--- Backups/pr3/RAPID/TASK1/PROGMOD/Module1.mod ---
MODULE Module1
	CONST robtarget Target_10:=[[1359.914350434,189.052041228,1867.751078124],[0.28377426,-0.836118095,0.437820703,-0.169386341],[0,0,-3,0],[9E+09,9E+09,9E+09,9E+09,9E+09,9E+09]];
	CONST robtarget Target_20:=[[1359.914369628,120.392226788,1867.751087064],[0.283774546,-0.836118001,0.43782057,-0.169386668],[0,0,-3,0],[9E+09,9E+09,9E+09,9E+09,9E+09,9E+09]];
	CONST robtarget Target_30:=[[1359.914226872,120.392161677,1060.024906535],[0.283774755,-0.836117846,0.437820445,-0.169387409],[0,1,-3,0],[9E+09,9E+09,9E+09,9E+09,9E+09,9E+09]];
	CONST robtarget Target_40:=[[1288.339226949,142.88058846,1159.109938579],[0.283774905,-0.836117579,0.437820302,-0.169388845],[0,1,-3,0],[9E+09,9E+09,9E+09,9E+09,9E+09,9E+09]];
	CONST robtarget Target_50:=[[1288.339333488,142.880646916,1864.033074108],[0.283776583,-0.836117259,0.437818944,-0.169391124],[0,0,-3,0],[9E+09,9E+09,9E+09,9E+09,9E+09,9E+09]];
	CONST robtarget Target_60:=[[1396.622330981,211.05352138,1797.840056923],[0.283777308,-0.836116859,0.437818886,-0.169392034],[0,0,-3,0],[9E+09,9E+09,9E+09,9E+09,9E+09,9E+09]];
	CONST robtarget Target_70:=[[1225.907089757,47.887281808,1220.291013598],[0.283778703,-0.836117031,0.437817025,-0.169393657],[-1,1,-3,0],[9E+09,9E+09,9E+09,9E+09,9E+09,9E+09]];
	CONST robtarget Target_80:=[[1225.907079131,47.887238756,979.783968451],[0.283778643,-0.836116986,0.437817072,-0.169393858],[-1,1,-3,0],[9E+09,9E+09,9E+09,9E+09,9E+09,9E+09]];
	CONST robtarget Target_90:=[[1225.907179869,110.196868604,823.578395227],[0.283778412,-0.836116876,0.43781729,-0.169394225],[0,1,-4,0],[9E+09,9E+09,9E+09,9E+09,9E+09,9E+09]];
	CONST robtarget Target_100:=[[1035.260759077,110.196845363,823.578341268],[0.283778036,-0.836117118,0.437816894,-0.169394683],[0,1,-4,0],[9E+09,9E+09,9E+09,9E+09,9E+09,9E+09]];
	CONST robtarget Target_110:=[[1035.261060311,110.196778558,823.57799127],[0.341042108,-0.743784627,0.47971346,-0.316780217],[0,2,-4,0],[9E+09,9E+09,9E+09,9E+09,9E+09,9E+09]];
	CONST robtarget Target_120:=[[1035.2615814,110.19683868,823.577736078],[0.306762006,-0.695295218,0.550476721,-0.345596603],[0,3,-5,0],[9E+09,9E+09,9E+09,9E+09,9E+09,9E+09]];
	CONST robtarget Target_130:=[[1227.749003758,-87.086102015,898.637389106],[0.401803093,-0.83564632,0.29691234,-0.228237957],[-1,1,-4,0],[9E+09,9E+09,9E+09,9E+09,9E+09,9E+09]];
	CONST robtarget Target_140:=[[1247.926834673,-113.238805252,518.057828259],[0.401801987,-0.835647129,0.296911763,-0.228237691],[-1,2,-4,0],[9E+09,9E+09,9E+09,9E+09,9E+09,9E+09]];
	CONST robtarget Target_150:=[[1264.237758862,-145.855770141,241.966431846],[0.401801453,-0.835648597,0.296909613,-0.228236053],[-1,2,-4,0],[9E+09,9E+09,9E+09,9E+09,9E+09,9E+09]];
	CONST robtarget Target_160:=[[1128.0688239,-143.135341759,292.908969476],[0.401800911,-0.835651508,0.296904199,-0.228233393],[-1,2,-4,0],[9E+09,9E+09,9E+09,9E+09,9E+09,9E+09]];
	CONST robtarget Target_170:=[[1128.069049024,-143.135368985,729.590033266],[0.401800633,-0.835651641,0.296904229,-0.228233356],[-1,1,-4,0],[9E+09,9E+09,9E+09,9E+09,9E+09,9E+09]];
	CONST robtarget Target_180:=[[1236.096802902,-96.606788938,264.050379664],[0.844944992,-0.381876574,0.080734356,-0.365677736],[-1,1,-4,1],[9E+09,9E+09,9E+09,9E+09,9E+09,9E+09]];
	CONST robtarget Target_190:=[[1263.432163062,-49.076157559,219.686861759],[0.84494253,-0.381881448,0.080736569,-0.365677845],[-1,1,-4,1],[9E+09,9E+09,9E+09,9E+09,9E+09,9E+09]];
	CONST robtarget Target_200:=[[1237.348016113,-55.067728806,185.37023784],[0.844936834,-0.381892704,0.080740996,-0.365678275],[-1,1,-4,1],[9E+09,9E+09,9E+09,9E+09,9E+09,9E+09]];
	CONST robtarget Target_210:=[[1065.206110583,-52.115045672,185.369462943],[0.844935801,-0.38189476,0.080741711,-0.365678357],[-1,1,-4,1],[9E+09,9E+09,9E+09,9E+09,9E+09,9E+09]];
	CONST robtarget Target_220:=[[1218.03502948,-52.114690425,166.267960314],[0.844934253,-0.381898356,0.080742219,-0.365678066],[-1,1,-4,1],[9E+09,9E+09,9E+09,9E+09,9E+09,9E+09]];
	CONST robtarget Target_230:=[[1218.035057782,0.360283476,166.267597723],[0.844933777,-0.381899344,0.08074267,-0.365678035],[-1,1,-4,1],[9E+09,9E+09,9E+09,9E+09,9E+09,9E+09]];
	CONST robtarget Target_240:=[[1049.013112504,0.360320531,166.267173862],[0.844933246,-0.381900492,0.080742991,-0.365677991],[-1,1,-4,1],[9E+09,9E+09,9E+09,9E+09,9E+09,9E+09]];
	CONST robtarget Target_250:=[[741.479498812,21.487944281,460.641074795],[0.167046833,0.579624718,0.293347911,0.741672127],[-1,2,-5,1],[9E+09,9E+09,9E+09,9E+09,9E+09,9E+09]];
	CONST robtarget Target_260:=[[741.47959356,52.990017017,468.573399202],[0.167047709,0.579627016,0.293349084,0.741669671],[0,2,-5,1],[9E+09,9E+09,9E+09,9E+09,9E+09,9E+09]];
	CONST robtarget Target_270:=[[741.479470826,52.989743441,402.945757804],[0.167048259,0.579628065,0.293349195,0.741668683],[0,2,-5,1],[9E+09,9E+09,9E+09,9E+09,9E+09,9E+09]];
	CONST robtarget Target_280:=[[741.479437654,-21.578976222,402.945438683],[0.167047992,0.579628558,0.293349684,0.741668165],[-1,2,-5,1],[9E+09,9E+09,9E+09,9E+09,9E+09,9E+09]];
	CONST robtarget Target_290:=[[741.479455644,-21.579005192,495.449003725],[0.167047914,0.579629056,0.29334997,0.74166768],[-1,2,-5,1],[9E+09,9E+09,9E+09,9E+09,9E+09,9E+09]];
	CONST robtarget Target_300:=[[954.088201372,127.514709299,272.759250433],[0.167048682,0.579633756,0.293351441,0.741663252],[0,2,-5,1],[9E+09,9E+09,9E+09,9E+09,9E+09,9E+09]];
	CONST robtarget Target_310:=[[954.088095411,127.514510621,-13.446080114],[0.167048969,0.579635488,0.293351958,0.741661629],[0,2,-5,1],[9E+09,9E+09,9E+09,9E+09,9E+09,9E+09]];
	CONST robtarget Target_320:=[[954.087987294,42.729988075,-13.446422439],[0.167048805,0.579636058,0.293352405,0.741661043],[-1,2,-5,1],[9E+09,9E+09,9E+09,9E+09,9E+09,9E+09]];
	CONST robtarget Target_330:=[[954.087890772,42.72997271,305.664990545],[0.167048406,0.579637688,0.293353566,0.741659401],[-1,2,-5,1],[9E+09,9E+09,9E+09,9E+09,9E+09,9E+09]];
	CONST robtarget Target_340:=[[1062.705954522,42.729934145,305.664692576],[0.167048487,0.579638189,0.293353947,0.74165884],[-1,2,-5,1],[9E+09,9E+09,9E+09,9E+09,9E+09,9E+09]];
	CONST robtarget Target_350:=[[1062.705913046,42.729918606,-20.939554836],[0.167048412,0.579638718,0.293354285,0.74165831],[-1,2,-5,1],[9E+09,9E+09,9E+09,9E+09,9E+09,9E+09]];
	CONST robtarget Target_360:=[[1062.705922672,-42.780840866,-20.939905277],[0.167048299,0.579639297,0.293354716,0.741657712],[-1,2,-5,1],[9E+09,9E+09,9E+09,9E+09,9E+09,9E+09]];
	CONST robtarget Target_370:=[[1062.705963822,-42.780859644,358.539699735],[0.167048216,0.579639878,0.293354953,0.741657182],[-1,2,-5,0],[9E+09,9E+09,9E+09,9E+09,9E+09,9E+09]];
	PERS num ColorIndex3:=1;
    CONST robtarget Target_180_2:=[[1236.09620943,-229.253997693,264.04805571],[0.892729073,-0.435461507,-0.046433543,-0.10607546],[-1,1,-4,1],[9E+09,9E+09,9E+09,9E+09,9E+09,9E+09]];
    CONST robtarget Target_380:=[[1062.706013298,254.661882488,394.279567264],[0.022239678,-0.602825102,-0.047180566,-0.79616662],[0,2,-5,1],[9E+09,9E+09,9E+09,9E+09,9E+09,9E+09]];
    CONST robtarget Target_390:=[[729.42291728,228.831924059,394.278056221],[0.022236675,-0.602828487,-0.047179166,-0.796164224],[0,2,-5,1],[9E+09,9E+09,9E+09,9E+09,9E+09,9E+09]];
    CONST robtarget Target_400:=[[992.762340696,228.831189854,180.25404409],[0.022234595,-0.602832885,-0.047178666,-0.796160982],[0,2,-5,1],[9E+09,9E+09,9E+09,9E+09,9E+09,9E+09]];
    CONST robtarget Target_410:=[[992.76307458,129.831933881,781.600340796],[0.005972285,-0.914865356,0.069810272,-0.397633295],[0,3,-6,0],[9E+09,9E+09,9E+09,9E+09,9E+09,9E+09]];
    CONST robtarget Target_420:=[[1274.891703819,171.05584658,1014.941903815],[0.005970392,-0.91486556,0.069814373,-0.397632135],[0,4,-6,0],[9E+09,9E+09,9E+09,9E+09,9E+09,9E+09]];
    CONST robtarget Target_430:=[[1047.127100193,89.200489047,835.063488807],[0.001681943,0.952786124,-0.070049154,0.295446931],[0,4,-7,0],[9E+09,9E+09,9E+09,9E+09,9E+09,9E+09]];
    PROC Path_10()
        ColorIndex3:=1;
        Set do3;
        WaitTime 1;
	    MoveL Target_10,v500,fine,tool0\WObj:=wobj0;
	    MoveL Target_20,v500,fine,tool0\WObj:=wobj0;
	    MoveL Target_30,v500,fine,tool0\WObj:=wobj0;
	    MoveL Target_40,v500,fine,tool0\WObj:=wobj0;
	    MoveL Target_50,v500,fine,tool0\WObj:=wobj0;
	    MoveL Target_60,v500,fine,tool0\WObj:=wobj0;
	    MoveL Target_70,v500,fine,tool0\WObj:=wobj0;
	    MoveL Target_80,v500,fine,tool0\WObj:=wobj0;
	    MoveL Target_90,v500,fine,tool0\WObj:=wobj0;
	    MoveL Target_100,v500,fine,tool0\WObj:=wobj0;
	    MoveL Target_110,v500,fine,tool0\WObj:=wobj0;
	    MoveL Target_120,v500,fine,tool0\WObj:=wobj0;
	    MoveL Target_130,v500,fine,tool0\WObj:=wobj0;
	    MoveL Target_140,v500,fine,tool0\WObj:=wobj0;
	    MoveL Target_150,v500,fine,tool0\WObj:=wobj0;
	    MoveL Target_160,v500,fine,tool0\WObj:=wobj0;
	    MoveL Target_170,v500,fine,tool0\WObj:=wobj0;
	    MoveL Target_180,v500,fine,tool0\WObj:=wobj0;
	    MoveL Target_180_2,v500,fine,tool0\WObj:=wobj0;
	    MoveL Target_180,v500,fine,tool0\WObj:=wobj0;
	    MoveL Target_190,v500,fine,tool0\WObj:=wobj0;
	    MoveL Target_200,v500,fine,tool0\WObj:=wobj0;
	    MoveL Target_210,v500,fine,tool0\WObj:=wobj0;
	    MoveL Target_220,v500,fine,tool0\WObj:=wobj0;
	    MoveL Target_230,v500,fine,tool0\WObj:=wobj0;
	    MoveL Target_240,v500,fine,tool0\WObj:=wobj0;
	    MoveL Target_250,v500,fine,tool0\WObj:=wobj0;
	    MoveL Target_260,v500,fine,tool0\WObj:=wobj0;
	    MoveL Target_270,v500,fine,tool0\WObj:=wobj0;
	    MoveL Target_280,v500,fine,tool0\WObj:=wobj0;
	    MoveL Target_290,v500,fine,tool0\WObj:=wobj0;
	    MoveL Target_310,v500,fine,tool0\WObj:=wobj0;
	    MoveL Target_320,v500,fine,tool0\WObj:=wobj0;
	    MoveL Target_330,v500,fine,tool0\WObj:=wobj0;
	    MoveL Target_350,v500,fine,tool0\WObj:=wobj0;
	    MoveL Target_360,v500,fine,tool0\WObj:=wobj0;
	    MoveL Target_370,v500,fine,tool0\WObj:=wobj0;
        MoveL Target_380,v500,fine,tool0\WObj:=wobj0;
        MoveL Target_390,v500,fine,tool0\WObj:=wobj0;
        MoveL Target_400,v1000,z100,tool0\WObj:=wobj0;
        MoveL Target_410,v1000,z100,tool0\WObj:=wobj0;
        MoveL Target_420,v1000,fine,tool0\WObj:=wobj0;
        MoveL Target_430,v1000,fine,tool0\WObj:=wobj0;
        WaitTime 1;
        Reset do3;
	ENDPROC
ENDMODULE

--- Backups/pr1/HOME/programs/calpos.mod ---
module calpos

   ! SCOPE: Universal calibration/sync position program.

   proc mainCalPos()
      var jointtarget jLocalCalPos;

      ! Dummy instruction for SetPP.
      WaitTime 1;

      ! Set default values for all axis.
      jLocalCalPos := [[9E+09,9E+09,9E+09,9E+09,9E+09,9E+09],[9E+09,9E+09,9E+09,9E+09,9E+09,0]];

      jLocalCalPos.robax.rax_1 := nArmCalPos("rob1_1");
      jLocalCalPos.robax.rax_2 := nArmCalPos("rob1_2");
      jLocalCalPos.robax.rax_3 := nArmCalPos("rob1_3");
      jLocalCalPos.robax.rax_4 := nArmCalPos("rob1_4");
      jLocalCalPos.robax.rax_5 := nArmCalPos("rob1_5");
      jLocalCalPos.robax.rax_6 := nArmCalPos("rob1_6");

      if nRobSerialPart() = 5500 or nRobSerialPart() = 5510 then
         ! IRB5500 and IRB5510 has special values on axis 5 and 6, just set to 0 as stated in the manual.
         jLocalCalPos.robax.rax_5 := 0;
         jLocalCalPos.robax.rax_6 := 0;
      endif

      if stSingleJoint("AX7_1") <> "" then
         ! 7-axis robot.
         jLocalCalPos.extax.eax_a := nArmCalPos(stSingleJoint("AX7_1") \NoConversion)*1000;
      elseif nArmCalPos("obp_3") <> 9E+09 then
         ! 3-axis TurnTable.
         !IndReset OBP,2\RefNum:=0\Short;
         !IndReset OBP,3\RefNum:=0\Short;
         jLocalCalPos.extax.eax_a := nArmCalPos("obp_1");
         jLocalCalPos.extax.eax_b := nArmCalPos("obp_2");
         jLocalCalPos.extax.eax_c := nArmCalPos("obp_3");
      elseif nArmCalPos("obp_2") <> 9E+09 then
         ! 2-axis TurnTable.
         jLocalCalPos.extax.eax_a := nArmCalPos("obp_1");
         jLocalCalPos.extax.eax_b := nArmCalPos("obp_2");
      elseif nArmCalPos("obp_1") <> 9E+09 then
         ! 1-axis TurnTable.
         jLocalCalPos.extax.eax_a := nArmCalPos("obp_1");
      elseif nArmCalPos("track1") <> 9E+09 then
         ! IRB5350-02.
         jLocalCalPos.robax.rax_4 := 0;
         jLocalCalPos.robax.rax_5 := 0;
         jLocalCalPos.robax.rax_6 := 0;
         jLocalCalPos.extax.eax_a := nArmCalPos("track1" \NoConversion);
      elseif stRobotType() = "ROB1_5350_01_T00F82_A21C21D21" then
         ! IRB5350-01.
         jLocalCalPos.robax.rax_4 := 0;
         jLocalCalPos.robax.rax_5 := 0;
         jLocalCalPos.robax.rax_6 := 0;
      else
         ! Attempt to get values for 8-axis robot.
         jLocalCalPos.extax.eax_a := nArmCalPos("rob1_7" \NoConversion);
         jLocalCalPos.extax.eax_b := nArmCalPos("rob1_8" \NoConversion);
      endif

      if stSingleJoint("H1AngleAxis") <> "" then
         ! Global CBS.
         jLocalCalPos.extax.eax_b := 0;
         jLocalCalPos.extax.eax_c := 0;
         jLocalCalPos.extax.eax_d := 0;
         jLocalCalPos.extax.eax_e := 0;
      endif

      MoveAbsJ jLocalCalPos,v100,fine,tool0;
      Stop;
   endproc

   local func num nArmCalPos(string stArm \switch NoConversion)
      var num nCalPos;
      ReadCfgData "/MOC/ARM/" + stArm, "cal_position", nCalPos;
      if Present(NoConversion) then
         return nCalPos;
      else
         return Round(nCalPos * (180 / 3.1415926) \Dec := 3);
      endif
   error
      if errno = ERR_CFG_NOTFND then
         SkipWarn;
         return 9E+09;
      endif
   endfunc

   local func string stSingleJoint(string stSingle)
      var string stJoint;
      ReadCfgData "/MOC/SINGLE/" + stSingle, "use_joint", stJoint;
      return stJoint;
   error
      if errno = ERR_CFG_NOTFND then
         SkipWarn;
         return "";
      endif
   endfunc

   local func num nRobSerialPart()
      var string stPart;
      var num nPart;
      ReadCfgData "/MOC/ROBOT_SERIAL_NUMBER/PID", "robot_serial_number_high_part", stPart;
      if StrToVal(StrPart(stPart, 1, StrFind(stPart, 1, "_") - 1), nPart) then
         return nPart;
      else
         return 9E+09;
      endif
   error
      SkipWarn;
      return 9E+09;
   endfunc

   local func string stRobotType()
      var string stType;
      ReadCfgData "/MOC/ROBOT/ROB_1", "use_robot_type", stType;
      return stType;
   error
      if errno = ERR_CFG_NOTFND then
         SkipWarn;
         return "";
      endif
   endfunc

endmodule

--- Backups/pr1/HOME/programs/m1.mod ---
MODULE M1

  PROC mainM1()
    WaitTime 10;
  ENDPROC

ENDMODULE

--- Backups/pr1/HOME/programs/m10001.mod ---
module m10001

   ! SCOPE: Motion program for home position.

   proc mainm10001()
      if jHomePos.robax.rax_1 = 9E+09 then
         ErrWrite \W, "Home position not taught!", "";
      else
         MoveAbsJ jHomePos,v300,fine,tUserTool0;
      endif
   endproc

endmodule

--- Backups/pr1/HOME/programs/m2.mod ---
MODULE M2

  PROC mainM2()
    WaitTime 10;
  ENDPROC

ENDMODULE

--- Backups/pr1/HOME/programs/m3.mod ---
MODULE M3

  PROC mainM3()
    WaitTime 10;
  ENDPROC

ENDMODULE

--- Backups/pr1/SYSPAR/EIO.cfg ---
EIO:CFG_1.0:6:1::
#
SYSSIG_OUT:

      -Status "AutoOn" -Signal "AutoModeOn"

      -Status "RunchOk" -Signal "RunChainClosed"

      -Status "Error" -Signal "sdoRobotError"

      -Status "CycleOn" -Signal "sdoCycleOn"

      -Status "EmStop" -Signal "EmergencyStop"

      -Status "MotOnState" -Signal "MotorIsOn"

      -Status "WriteAccess" -Signal "MasterGranted"

      -Status "MotSupTrigg" -Signal "MotionSupTrigg"
#
SYSSIG_IN:

      -Signal "sdoAckAutoMode" -Action "AckAutoMode"

      -Signal "sdoResetError" -Action "ResetError"

      -Signal "sdoStartMain" -Action "StartMain"

      -Signal "sdoMotOnStart" -Action "MotOnStart"

      -Signal "sdoStop" -Action "Stop"

      -Signal "sdoQuickStop" -Action "QuickStop"

      -Signal "sdoMotorOn" -Action "MotorOn"

      -Signal "sdoMotorOff" -Action "MotorOff"

      -Signal "sdoWriteRequest" -Action "WriteAccess"
#
INDUSTRIAL_NETWORK:

      -Name "DeviceNet" -Label "DeviceNet Master/Slave Network" -Address "2"
#
EIO_CROSS:

      -Name "ReadyToReceiveCross" -Res "ReadyToReceive" -Act1 "doQueueFull"\
      -Act1_invert

      -Name "JobPendingCross" -Res "JobPending" -Act1 "doQueueEmpty"\
      -Act1_invert

      -Name "MtrlChRunningCross" -Res "MtrlChRunning" -Act1 "doMCSuspended"\
      -Act1_invert

      -Name "AppEnabledCross" -Res "AppEnabled" -Act1 "A1Enable"

      -Name "AppErrorCross" -Res "AppError" -Act1 "A1Error"

      -Name "HVEnabledCross" -Res "HVEnabled" -Act1 "A1HVEn" -Oper1 "AND"\
      -Act2 "READY_HV_ON"

      -Name "PotLifeWarningCross" -Res "PotLifeWarning" -Act1 "A1FluidPlWS"

      -Name "PotLifeTimeOutCross" -Res "PotLifeTimeOut" -Act1 "A1FluidPlTO"

      -Name "HomePosCross" -Res "HomePos" -Act1 "doHomePos"

      -Name "MtrlChangePosCross" -Res "MtrlChangePos" -Act1 "doMtrlChangePos"

      -Name "ReadyPosCross" -Res "ReadyPos" -Act1 "doReadyPos"

      -Name "UserPosCross" -Res "UserPos" -Act1 "doUserPos"

      -Name "doSwitchInAutoCross" -Res "doSwitchInAuto" -Act1 "AUTO1"\
      -Oper1 "AND" -Act2 "AUTO2"

      -Name "GoingToAutoCross" -Res "GoingToAuto" -Act1 "doSwitchInAuto"\
      -Oper1 "AND" -Act2 "AutoModeOn" -Act2_invert

      -Name "ReadyHighPriCross" -Res "ReadyHighPri" -Act1 "sdoCycleOn"\
      -Oper1 "AND" -Act2 "JobInProgress" -Act2_invert

      -Name "SystemRunningCross" -Res "SystemRunning" -Act1 "sdoCycleOn"\
      -Oper1 "AND" -Act2 "doQueuePause" -Act2_invert

      -Name "RobotErrorCross" -Res "RobotError" -Act1 "sdoRobotError"\
      -Oper1 "OR" -Act2 "doPntRapidError"

      -Name "BellRotatingCross" -Res "BellRotating" -Act1 "A1BellRotating"
#
DEVICENET_INTERNAL_DEVICE:

      -Name "DN_Internal_Device" -VendorName "ABB Robotics"\
      -ProductName "DeviceNet Internal Slave Device"
#
ICI_DEVICE:

      -Name "PIB" -Network "ICI" -Label "Process Interface Board"\
      -Address "192.168.126.200"
#
EIO_SIGNAL:

      -Name "AutoModeOn" -SignalType "DO"

      -Name "MasterGranted" -SignalType "DO"

      -Name "RunChainClosed" -SignalType "DO"

      -Name "RobotError" -SignalType "DO"

      -Name "JobInProgress" -SignalType "DO"

      -Name "JobPending" -SignalType "DO"

      -Name "ReadyHighPri" -SignalType "DO"

      -Name "SystemRunning" -SignalType "DO"

      -Name "MtrlChRunning" -SignalType "DO"

      -Name "MtrlChangeOn" -SignalType "DO"

      -Name "ObjConnected" -SignalType "DO"

      -Name "MtrlSupplyError" -SignalType "DO"

      -Name "AppEnabled" -SignalType "DO"

      -Name "AppError" -SignalType "DO"

      -Name "HVEnabled" -SignalType "DO"

      -Name "HVError" -SignalType "DO"

      -Name "PotLifeWarning" -SignalType "DO"

      -Name "PotLifeTimeOut" -SignalType "DO"

      -Name "HomePos" -SignalType "DO"

      -Name "MtrlChangePos" -SignalType "DO"

      -Name "ReadyPos" -SignalType "DO"

      -Name "UserPos" -SignalType "DO"

      -Name "ReposFinished" -SignalType "DO"

      -Name "EmergencyStop" -SignalType "DO"

      -Name "JobComplete" -SignalType "DO"

      -Name "GoingToAuto" -SignalType "DO"

      -Name "ReadyToReceive" -SignalType "DO"

      -Name "MotorIsOn" -SignalType "DO"

      -Name "ConveyorRunning" -SignalType "DO"

      -Name "ProgramLoaded" -SignalType "DO"

      -Name "CBSMotorIsOn" -SignalType "DO"

      -Name "BellRotating" -SignalType "DO"

      -Name "MotionSupTrigg" -SignalType "DO"

      -Name "doQueueFull" -SignalType "DO"

      -Name "doQueueEmpty" -SignalType "DO"

      -Name "doQueuePause" -SignalType "DO"

      -Name "doInModule" -SignalType "DO"

      -Name "doMCSuspended" -SignalType "DO"

      -Name "A1Enable" -SignalType "DO" -Access "All"

      -Name "A1Error" -SignalType "DO" -Access "All"

      -Name "A1HVEn" -SignalType "DO" -Access "All"

      -Name "A1FluidPlWS" -SignalType "DO" -Access "All"

      -Name "A1FluidPlTO" -SignalType "DO" -Access "All"

      -Name "doHomePos" -SignalType "DO" -Access "ReadOnly"

      -Name "doMtrlChangePos" -SignalType "DO" -Access "ReadOnly"

      -Name "doReadyPos" -SignalType "DO" -Access "ReadOnly"

      -Name "doUserPos" -SignalType "DO" -Access "ReadOnly"

      -Name "doSwitchInAuto" -SignalType "DO"

      -Name "doPntRapidError" -SignalType "DO"

      -Name "sdoRobotError" -SignalType "DO"

      -Name "sdoAckAutoMode" -SignalType "DO"

      -Name "sdoResetError" -SignalType "DO"

      -Name "sdoStartMain" -SignalType "DO"

      -Name "sdoMotOnStart" -SignalType "DO"

      -Name "sdoStop" -SignalType "DO"

      -Name "sdoQuickStop" -SignalType "DO"

      -Name "sdoMotorOn" -SignalType "DO"

      -Name "sdoMotorOff" -SignalType "DO"

      -Name "sdoCycleOn" -SignalType "DO"

      -Name "sdoWriteRequest" -SignalType "DO"

      -Name "A1Brush" -SignalType "GO" -Access "All"

      -Name "A1BrushTabNdx" -SignalType "GO" -Access "All"

      -Name "A1HVErrNo" -SignalType "GO" -Access "All"

      -Name "A1Material" -SignalType "GO" -Access "All"

      -Name "A1Fluid" -SignalType "AO" -Access "All"

      -Name "A1FluidAccu" -SignalType "AO" -Access "All"

      -Name "A1FluidEn" -SignalType "DO" -Access "All"

      -Name "A1NeedleEn" -SignalType "DO" -Access "All"

      -Name "A1BellRotating" -SignalType "DI" -Access "All"

      -Name "A1BrushTabLimEn" -SignalType "DO" -Access "All"

      -Name "do1" -SignalType "DO"

--- Backups/pr1/SYSPAR/PROC.cfg ---
PROC:CFG_1.0:6:0::
#
PW_SYSTEM:

      -name "PW_SYS" -pw_function "PW_FUNC"
#
PW_FUNCTION:

      -name "PW_FUNC" -do_repos_finished "ReposFinished"
#
PW_SERVICES_CONFIG:

      -Name "ProgramDirectory" -Value "HOME:/programs/"

      -Name "ProgramCache" -Value "False"

      -Name "LoadFailureModule" -Value ""

      -Name "ProgramStaticLoad" -Value "False"

      -Name "ProgramBackupSave" -Value "False"

      -Name "ProdLogDirectory" -Value "HOME:/logs"

      -Name "ProdLogFormat"\
      -Value "%D,Prog:%P,Mtrl:%M,Brush:%B,Usage:%C,CycleTime:%T"

      -Name "ProdLogSize" -Value "100000"

      -Name "JobQueueSize" -Value "10"

      -Name "JobQueueSave" -Value "False"

      -Name "JobQueueExpediteBegin" -Value "10001"

      -Name "JobQueueExpediteEnd" -Value "10016"

      -Name "ProgramIndexFile" -Value "HOME:/programs/segments.ndx"

      -Name "ExternalStart" -Value "False"

      -Name "JobQueueIgnoreMaterial" -Value "True"

      -Name "TipCleanModule" -Value "TipClean"

      -Name "TipCleanInterval" -Value "0"

      -Name "TipCleanModuleFile" -Value ""

      -Name "TipCleanIntervalFile" -Value ""

      -Name "AppCleanModule" -Value "AppClean"

      -Name "AppCleanInterval" -Value "0"

      -Name "AppCleanModuleFile" -Value ""

      -Name "AppCleanIntervalFile" -Value ""

      -Name "AppCleanHasPriority" -Value "False"

      -Name "BrushMapFormula" -Value "M"

      -Name "BrushMapFilter" -Value "999999"

      -Name "BrushMapZeroDefault" -Value "0"

      -Name "HVAckSignal" -Value "HV_ILCK_ACK"

      -Name "HVAckDelay" -Value "200"

      -Name "A1EnableSignal" -Value "A1Enable"

      -Name "A1ErrorSignal" -Value "A1Error"

      -Name "A1BrushTabNdxSignal" -Value "A1BrushTabNdx"

      -Name "A1BrushTabLimEnSignal" -Value "A1BrushTabLimEn"

      -Name "A1FluidAccuSignal" -Value "A1FluidAccu"

      -Name "A1HVEnSignal" -Value "A1HVEn"

      -Name "A1HVErrNoSignal" -Value "A1HVErrNo"

      -Name "A1BrushDevice" -Value "A1Brush"

      -Name "A1FluidEnSignal" -Value "A1FluidEn"

      -Name "A1NeedleEnSignal" -Value "A1NeedleEn"

      -Name "A1MaterialSignal" -Value "A1Material"

      -Name "CmdLogDirectory" -Value "HOME:/logs"

      -Name "CmdLogSize" -Value "100000"

      -Name "RobotDataDirectory" -Value "HOME:/robdata/"

      -Name "ProgramAliasFile" -Value "HOME:/alias/program.map"

      -Name "MaterialAliasFile" -Value "HOME:/alias/material.map"

      -Name "OptionAliasFile" -Value "HOME:/alias/option.map"
#
PW_EVENT_HOOKS:

      -Routine "TipCleanPreMain" -Event "PRE_MAIN" -Priority 55

      -Routine "TipCleanPostMain" -Event "POST_MAIN" -Priority 75

      -Routine "PreMainPosMsg" -Event "PRE_MAIN" -Priority 80

      -Routine "PostMainPosMsg" -Event "POST_MAIN" -Priority 20

      -Routine "PreMainCustom" -Event "PRE_MAIN"

      -Routine "PostMainCustom" -Event "POST_MAIN"
#
PW_SIGNAL_OUT:

      -Status "Resource:Loop.InJob" -Signal "JobInProgress"

      -Status "Resource:Loop.InModule" -Signal "doInModule"

      -Status "Resource:Loop.ProgramLoaded" -Signal "ProgramLoaded"

      -Status "Resource:Queue.Empty" -Signal "doQueueEmpty"

      -Status "Resource:Queue.Inhibited" -Signal "doQueuePause"

      -Status "Resource:MCEngine.Suspended" -Signal "doMCSuspended"

      -Status "Resource:MCEngine.On" -Signal "MtrlChangeOn"

      -Status "Resource:MCLog.ErrorStatus" -Signal "MtrlSupplyError"

      -Status "Resource:Queue.Full" -Signal "doQueueFull"

      -Status "Resource:App.HVError" -Signal "HVError"

--- Backups/pr2/SYSPAR/EIO.cfg ---
EIO:CFG_1.0:6:1::
#
SYSSIG_OUT:

      -Status "AutoOn" -Signal "AutoModeOn"

      -Status "RunchOk" -Signal "RunChainClosed"

      -Status "Error" -Signal "sdoRobotError"

      -Status "CycleOn" -Signal "sdoCycleOn"

      -Status "EmStop" -Signal "EmergencyStop"

      -Status "MotOnState" -Signal "MotorIsOn"

      -Status "WriteAccess" -Signal "MasterGranted"

      -Status "MotSupTrigg" -Signal "MotionSupTrigg"
#
SYSSIG_IN:

      -Signal "sdoAckAutoMode" -Action "AckAutoMode"

      -Signal "sdoResetError" -Action "ResetError"

      -Signal "sdoStartMain" -Action "StartMain"

      -Signal "sdoMotOnStart" -Action "MotOnStart"

      -Signal "sdoStop" -Action "Stop"

      -Signal "sdoQuickStop" -Action "QuickStop"

      -Signal "sdoMotorOn" -Action "MotorOn"

      -Signal "sdoMotorOff" -Action "MotorOff"

      -Signal "sdoWriteRequest" -Action "WriteAccess"
#
INDUSTRIAL_NETWORK:

      -Name "DeviceNet" -Label "DeviceNet Master/Slave Network" -Address "2"
#
EIO_CROSS:

      -Name "ReadyToReceiveCross" -Res "ReadyToReceive" -Act1 "doQueueFull"\
      -Act1_invert

      -Name "JobPendingCross" -Res "JobPending" -Act1 "doQueueEmpty"\
      -Act1_invert

      -Name "MtrlChRunningCross" -Res "MtrlChRunning" -Act1 "doMCSuspended"\
      -Act1_invert

      -Name "AppEnabledCross" -Res "AppEnabled" -Act1 "A1Enable"

      -Name "AppErrorCross" -Res "AppError" -Act1 "A1Error"

      -Name "HVEnabledCross" -Res "HVEnabled" -Act1 "A1HVEn" -Oper1 "AND"\
      -Act2 "READY_HV_ON"

      -Name "PotLifeWarningCross" -Res "PotLifeWarning" -Act1 "A1FluidPlWS"

      -Name "PotLifeTimeOutCross" -Res "PotLifeTimeOut" -Act1 "A1FluidPlTO"

      -Name "HomePosCross" -Res "HomePos" -Act1 "doHomePos"

      -Name "MtrlChangePosCross" -Res "MtrlChangePos" -Act1 "doMtrlChangePos"

      -Name "ReadyPosCross" -Res "ReadyPos" -Act1 "doReadyPos"

      -Name "UserPosCross" -Res "UserPos" -Act1 "doUserPos"

      -Name "doSwitchInAutoCross" -Res "doSwitchInAuto" -Act1 "AUTO1"\
      -Oper1 "AND" -Act2 "AUTO2"

      -Name "GoingToAutoCross" -Res "GoingToAuto" -Act1 "doSwitchInAuto"\
      -Oper1 "AND" -Act2 "AutoModeOn" -Act2_invert

      -Name "ReadyHighPriCross" -Res "ReadyHighPri" -Act1 "sdoCycleOn"\
      -Oper1 "AND" -Act2 "JobInProgress" -Act2_invert

      -Name "SystemRunningCross" -Res "SystemRunning" -Act1 "sdoCycleOn"\
      -Oper1 "AND" -Act2 "doQueuePause" -Act2_invert

      -Name "RobotErrorCross" -Res "RobotError" -Act1 "sdoRobotError"\
      -Oper1 "OR" -Act2 "doPntRapidError"

      -Name "BellRotatingCross" -Res "BellRotating" -Act1 "A1BellRotating"
#
DEVICENET_INTERNAL_DEVICE:

      -Name "DN_Internal_Device" -VendorName "ABB Robotics"\
      -ProductName "DeviceNet Internal Slave Device"
#
ICI_DEVICE:

      -Name "PIB" -Network "ICI" -Label "Process Interface Board"\
      -Address "192.168.126.200"
#
EIO_SIGNAL:

      -Name "AutoModeOn" -SignalType "DO"

      -Name "MasterGranted" -SignalType "DO"

      -Name "RunChainClosed" -SignalType "DO"

      -Name "RobotError" -SignalType "DO"

      -Name "JobInProgress" -SignalType "DO"

      -Name "JobPending" -SignalType "DO"

      -Name "ReadyHighPri" -SignalType "DO"

      -Name "SystemRunning" -SignalType "DO"

      -Name "MtrlChRunning" -SignalType "DO"

      -Name "MtrlChangeOn" -SignalType "DO"

      -Name "ObjConnected" -SignalType "DO"

      -Name "MtrlSupplyError" -SignalType "DO"

      -Name "AppEnabled" -SignalType "DO"

      -Name "AppError" -SignalType "DO"

      -Name "HVEnabled" -SignalType "DO"

      -Name "HVError" -SignalType "DO"

      -Name "PotLifeWarning" -SignalType "DO"

      -Name "PotLifeTimeOut" -SignalType "DO"

      -Name "HomePos" -SignalType "DO"

      -Name "MtrlChangePos" -SignalType "DO"

      -Name "ReadyPos" -SignalType "DO"

      -Name "UserPos" -SignalType "DO"

      -Name "ReposFinished" -SignalType "DO"

      -Name "EmergencyStop" -SignalType "DO"

      -Name "JobComplete" -SignalType "DO"

      -Name "GoingToAuto" -SignalType "DO"

      -Name "ReadyToReceive" -SignalType "DO"

      -Name "MotorIsOn" -SignalType "DO"

      -Name "ConveyorRunning" -SignalType "DO"

      -Name "ProgramLoaded" -SignalType "DO"

      -Name "CBSMotorIsOn" -SignalType "DO"

      -Name "BellRotating" -SignalType "DO"

      -Name "MotionSupTrigg" -SignalType "DO"

      -Name "doQueueFull" -SignalType "DO"

      -Name "doQueueEmpty" -SignalType "DO"

      -Name "doQueuePause" -SignalType "DO"

      -Name "doInModule" -SignalType "DO"

      -Name "doMCSuspended" -SignalType "DO"

      -Name "A1Enable" -SignalType "DO" -Access "All"

      -Name "A1Error" -SignalType "DO" -Access "All"

      -Name "A1HVEn" -SignalType "DO" -Access "All"

      -Name "A1FluidPlWS" -SignalType "DO" -Access "All"

      -Name "A1FluidPlTO" -SignalType "DO" -Access "All"

      -Name "doHomePos" -SignalType "DO" -Access "ReadOnly"

      -Name "doMtrlChangePos" -SignalType "DO" -Access "ReadOnly"

      -Name "doReadyPos" -SignalType "DO" -Access "ReadOnly"

      -Name "doUserPos" -SignalType "DO" -Access "ReadOnly"

      -Name "doSwitchInAuto" -SignalType "DO"

      -Name "doPntRapidError" -SignalType "DO"

      -Name "sdoRobotError" -SignalType "DO"

      -Name "sdoAckAutoMode" -SignalType "DO"

      -Name "sdoResetError" -SignalType "DO"

      -Name "sdoStartMain" -SignalType "DO"

      -Name "sdoMotOnStart" -SignalType "DO"

      -Name "sdoStop" -SignalType "DO"

      -Name "sdoQuickStop" -SignalType "DO"

      -Name "sdoMotorOn" -SignalType "DO"

      -Name "sdoMotorOff" -SignalType "DO"

      -Name "sdoCycleOn" -SignalType "DO"

      -Name "sdoWriteRequest" -SignalType "DO"

      -Name "A1Brush" -SignalType "GO" -Access "All"

      -Name "A1BrushTabNdx" -SignalType "GO" -Access "All"

      -Name "A1HVErrNo" -SignalType "GO" -Access "All"

      -Name "A1Material" -SignalType "GO" -Access "All"

      -Name "A1Fluid" -SignalType "AO" -Access "All"

      -Name "A1FluidAccu" -SignalType "AO" -Access "All"

      -Name "A1FluidEn" -SignalType "DO" -Access "All"

      -Name "A1NeedleEn" -SignalType "DO" -Access "All"

      -Name "A1BellRotating" -SignalType "DI" -Access "All"

      -Name "A1BrushTabLimEn" -SignalType "DO" -Access "All"

      -Name "do2" -SignalType "DO"

--- Backups/pr3/SYSPAR/EIO.cfg ---
EIO:CFG_1.0:6:1::
#
SYSSIG_OUT:

      -Status "AutoOn" -Signal "AutoModeOn"

      -Status "RunchOk" -Signal "RunChainClosed"

      -Status "Error" -Signal "sdoRobotError"

      -Status "CycleOn" -Signal "sdoCycleOn"

      -Status "EmStop" -Signal "EmergencyStop"

      -Status "MotOnState" -Signal "MotorIsOn"

      -Status "WriteAccess" -Signal "MasterGranted"

      -Status "MotSupTrigg" -Signal "MotionSupTrigg"
#
SYSSIG_IN:

      -Signal "sdoAckAutoMode" -Action "AckAutoMode"

      -Signal "sdoResetError" -Action "ResetError"

      -Signal "sdoStartMain" -Action "StartMain"

      -Signal "sdoMotOnStart" -Action "MotOnStart"

      -Signal "sdoStop" -Action "Stop"

      -Signal "sdoQuickStop" -Action "QuickStop"

      -Signal "sdoMotorOn" -Action "MotorOn"

      -Signal "sdoMotorOff" -Action "MotorOff"

      -Signal "sdoWriteRequest" -Action "WriteAccess"
#
INDUSTRIAL_NETWORK:

      -Name "DeviceNet" -Label "DeviceNet Master/Slave Network" -Address "2"
#
EIO_CROSS:

      -Name "ReadyToReceiveCross" -Res "ReadyToReceive" -Act1 "doQueueFull"\
      -Act1_invert

      -Name "JobPendingCross" -Res "JobPending" -Act1 "doQueueEmpty"\
      -Act1_invert

      -Name "MtrlChRunningCross" -Res "MtrlChRunning" -Act1 "doMCSuspended"\
      -Act1_invert

      -Name "AppEnabledCross" -Res "AppEnabled" -Act1 "A1Enable"

      -Name "AppErrorCross" -Res "AppError" -Act1 "A1Error"

      -Name "HVEnabledCross" -Res "HVEnabled" -Act1 "A1HVEn" -Oper1 "AND"\
      -Act2 "READY_HV_ON"

      -Name "PotLifeWarningCross" -Res "PotLifeWarning" -Act1 "A1FluidPlWS"

      -Name "PotLifeTimeOutCross" -Res "PotLifeTimeOut" -Act1 "A1FluidPlTO"

      -Name "HomePosCross" -Res "HomePos" -Act1 "doHomePos"

      -Name "MtrlChangePosCross" -Res "MtrlChangePos" -Act1 "doMtrlChangePos"

      -Name "ReadyPosCross" -Res "ReadyPos" -Act1 "doReadyPos"

      -Name "UserPosCross" -Res "UserPos" -Act1 "doUserPos"

      -Name "doSwitchInAutoCross" -Res "doSwitchInAuto" -Act1 "AUTO1"\
      -Oper1 "AND" -Act2 "AUTO2"

      -Name "GoingToAutoCross" -Res "GoingToAuto" -Act1 "doSwitchInAuto"\
      -Oper1 "AND" -Act2 "AutoModeOn" -Act2_invert

      -Name "ReadyHighPriCross" -Res "ReadyHighPri" -Act1 "sdoCycleOn"\
      -Oper1 "AND" -Act2 "JobInProgress" -Act2_invert

      -Name "SystemRunningCross" -Res "SystemRunning" -Act1 "sdoCycleOn"\
      -Oper1 "AND" -Act2 "doQueuePause" -Act2_invert

      -Name "RobotErrorCross" -Res "RobotError" -Act1 "sdoRobotError"\
      -Oper1 "OR" -Act2 "doPntRapidError"

      -Name "BellRotatingCross" -Res "BellRotating" -Act1 "A1BellRotating"
#
DEVICENET_INTERNAL_DEVICE:

      -Name "DN_Internal_Device" -VendorName "ABB Robotics"\
      -ProductName "DeviceNet Internal Slave Device"
#
ICI_DEVICE:

      -Name "PIB" -Network "ICI" -Label "Process Interface Board"\
      -Address "192.168.126.200"
#
EIO_SIGNAL:

      -Name "AutoModeOn" -SignalType "DO"

      -Name "MasterGranted" -SignalType "DO"

      -Name "RunChainClosed" -SignalType "DO"

      -Name "RobotError" -SignalType "DO"

      -Name "JobInProgress" -SignalType "DO"

      -Name "JobPending" -SignalType "DO"

      -Name "ReadyHighPri" -SignalType "DO"

      -Name "SystemRunning" -SignalType "DO"

      -Name "MtrlChRunning" -SignalType "DO"

      -Name "MtrlChangeOn" -SignalType "DO"

      -Name "ObjConnected" -SignalType "DO"

      -Name "MtrlSupplyError" -SignalType "DO"

      -Name "AppEnabled" -SignalType "DO"

      -Name "AppError" -SignalType "DO"

      -Name "HVEnabled" -SignalType "DO"

      -Name "HVError" -SignalType "DO"

      -Name "PotLifeWarning" -SignalType "DO"

      -Name "PotLifeTimeOut" -SignalType "DO"

      -Name "HomePos" -SignalType "DO"

      -Name "MtrlChangePos" -SignalType "DO"

      -Name "ReadyPos" -SignalType "DO"

      -Name "UserPos" -SignalType "DO"

      -Name "ReposFinished" -SignalType "DO"

      -Name "EmergencyStop" -SignalType "DO"

      -Name "JobComplete" -SignalType "DO"

      -Name "GoingToAuto" -SignalType "DO"

      -Name "ReadyToReceive" -SignalType "DO"

      -Name "MotorIsOn" -SignalType "DO"

      -Name "ConveyorRunning" -SignalType "DO"

      -Name "ProgramLoaded" -SignalType "DO"

      -Name "CBSMotorIsOn" -SignalType "DO"

      -Name "BellRotating" -SignalType "DO"

      -Name "MotionSupTrigg" -SignalType "DO"

      -Name "doQueueFull" -SignalType "DO"

      -Name "doQueueEmpty" -SignalType "DO"

      -Name "doQueuePause" -SignalType "DO"

      -Name "doInModule" -SignalType "DO"

      -Name "doMCSuspended" -SignalType "DO"

      -Name "A1Enable" -SignalType "DO" -Access "All"

      -Name "A1Error" -SignalType "DO" -Access "All"

      -Name "A1HVEn" -SignalType "DO" -Access "All"

      -Name "A1FluidPlWS" -SignalType "DO" -Access "All"

      -Name "A1FluidPlTO" -SignalType "DO" -Access "All"

      -Name "doHomePos" -SignalType "DO" -Access "ReadOnly"

      -Name "doMtrlChangePos" -SignalType "DO" -Access "ReadOnly"

      -Name "doReadyPos" -SignalType "DO" -Access "ReadOnly"

      -Name "doUserPos" -SignalType "DO" -Access "ReadOnly"

      -Name "doSwitchInAuto" -SignalType "DO"

      -Name "doPntRapidError" -SignalType "DO"

      -Name "sdoRobotError" -SignalType "DO"

      -Name "sdoAckAutoMode" -SignalType "DO"

      -Name "sdoResetError" -SignalType "DO"

      -Name "sdoStartMain" -SignalType "DO"

      -Name "sdoMotOnStart" -SignalType "DO"

      -Name "sdoStop" -SignalType "DO"

      -Name "sdoQuickStop" -SignalType "DO"

      -Name "sdoMotorOn" -SignalType "DO"

      -Name "sdoMotorOff" -SignalType "DO"

      -Name "sdoCycleOn" -SignalType "DO"

      -Name "sdoWriteRequest" -SignalType "DO"

      -Name "A1Brush" -SignalType "GO" -Access "All"

      -Name "A1BrushTabNdx" -SignalType "GO" -Access "All"

      -Name "A1HVErrNo" -SignalType "GO" -Access "All"

      -Name "A1Material" -SignalType "GO" -Access "All"

      -Name "A1Fluid" -SignalType "AO" -Access "All"

      -Name "A1FluidAccu" -SignalType "AO" -Access "All"

      -Name "A1FluidEn" -SignalType "DO" -Access "All"

      -Name "A1NeedleEn" -SignalType "DO" -Access "All"

      -Name "A1BellRotating" -SignalType "DI" -Access "All"

      -Name "A1BrushTabLimEn" -SignalType "DO" -Access "All"

      -Name "do3" -SignalType "DO"
